{attribute 'linkalways'} 
{attribute 'no_explicit_call' := 'This FB is a CLASS and must be accessed using methods or properties'}
{attribute 'enable_dynamic_creation'}
FUNCTION_BLOCK _ETcVnFeatureScoreTypeORB EXTENDS EnumDatatypeBase
VAR
	localData : ETcVnFeatureScoreTypeORB;
	activeData : REFERENCE TO ETcVnFeatureScoreTypeORB;
	enumBaseDatatype : _DINT(localData);
END_VAR

METHOD PRIVATE AddLocalEnumeration
VAR_INPUT
	Enumeration : T_MAXSTRING;
	Value : ETcVnFeatureScoreTypeORB;
END_VAR
AddEnumeration(Enumeration, Value);
END_METHOD

PROPERTY PUBLIC Address : PVOID
GET
Address := ADR(activeData);
END_GET
END_PROPERTY

METHOD PUBLIC ClearReference
VAR_INPUT
END_VAR
activeData REF= localData;
SetBaseDatatypeReference();
END_METHOD

METHOD PUBLIC Clone : I_Datatype
VAR
    pClone : POINTER TO _ETcVnFeatureScoreTypeORB;
END_VAR
pClone := __NEW(_ETcVnFeatureScoreTypeORB(InitialValue := Value));
Clone := pClone^;
END_METHOD

METHOD FB_init : BOOL
VAR_INPUT
	bInitRetains : BOOL; // if TRUE, the retain variables are initialized (warm start / cold start)
	bInCopyCode : BOOL;  // if TRUE, the instance afterwards gets moved into the copy code (online change)
	InitialValue : ETcVnFeatureScoreTypeORB;
END_VAR
localData := InitialValue;
AddBaseDatatype(enumBaseDatatype);
ClearReference();

AddLocalEnumeration('TCVN_FST_ORB_HARRIS', ETcVnFeatureScoreTypeORB.TCVN_FST_ORB_HARRIS);
AddLocalEnumeration('TCVN_FST_ORB_FAST', ETcVnFeatureScoreTypeORB.TCVN_FST_ORB_FAST);
END_METHOD

PROPERTY PUBLIC Identifier : T_MAXSTRING
GET
Identifier := 'ETcVnFeatureScoreTypeORB';
END_GET
END_PROPERTY

METHOD IsEnumeratorValueEqual : BOOL
VAR_INPUT
	Enumerator : I_KeyValueForwardEnumerator;
END_VAR
VAR
	storedValue : ETcVnFeatureScoreTypeORB;
END_VAR
IF NOT Enumerator.TryGet(storedValue) THEN
	RETURN;
END_IF

IsEnumeratorValueEqual := storedValue = activeData;
END_METHOD

METHOD PUBLIC MakeReferenceTo
VAR_INPUT
	ReferenceTarget : REFERENCE TO ETcVnFeatureScoreTypeORB;
END_VAR
activeData REF= ReferenceTarget;
SetBaseDatatypeReference();
END_METHOD

METHOD PROTECTED SetBaseDatatypeReference
VAR_INPUT
END_VAR
enumBaseDatatype.MakeReferenceTo(activeData);
END_METHOD

PROPERTY PUBLIC Size : UDINT
GET
Size := SIZEOF(activeData);
END_GET
END_PROPERTY

METHOD TryMakeReferenceTo : BOOL
VAR_INPUT
	Target : I_Datatype;
END_VAR
VAR
	targetAsEnum : I_EnumDatatype;
	pTargetData : POINTER TO ETcVnFeatureScoreTypeORB;
END_VAR
IF NOT Target.TryResolveAsEnumDatatype(targetAsEnum) THEN
	RETURN;
END_IF

IF targetAsEnum.Identifier <> Identifier THEN
	RETURN;
END_IF

pTargetData := Target.Address;
activeData REF= pTargetData^;
SetBaseDatatypeReference();
TryMakeReferenceTo := TRUE;
END_METHOD

PROPERTY PUBLIC Value : ETcVnFeatureScoreTypeORB
GET
Value := activeData;
END_GET
SET
activeData := Value;
END_SET
END_PROPERTY

END_FUNCTION_BLOCK

(* stored: Version 1.1.0.1, ProductVersion 3.1.4024.13
   POU _ETcVnFeatureScoreTypeORB: Id {15c0cc44-f562-0f51-0f9a-718f0dddc65b}, SpecialFunc None
   Folder Core: Id {df601a09-cbae-02db-08fe-8ac88da08644}
   Folder Protected: Id {92163e21-aa89-0321-267b-a355ab4cae68}
   Folder Customize: Id {6d3a5763-e8d1-0f13-33df-945d8160b9e1}
   Folder Constructor: Id {8b40bffe-e2be-0495-1321-7413e1ad65e8}
   Folder Private: Id {aa80153e-39fb-0732-36e3-7e3ad3f38d94}
   Folder Protected: Id {4633f427-e61f-0493-0688-5742aa9f23d0}
   Method AddLocalEnumeration: Id {9f39223e-9470-039e-39a8-0675ce62e4ff}
   Property Address: Id {6760ea54-2415-03cb-3177-bfceedc2a8c9}
   Get Get: Id {5bc95193-dc58-0e53-18da-11d1bd8a60da}
   Method ClearReference: Id {e3220401-e4c1-091b-0760-324778c8aa33}
   Method Clone: Id {64985a08-8ed4-0345-30e0-1f5738597027}
   Method FB_init: Id {4c1f1c28-98dc-0ef3-3dd7-6976fc278be2}
   Property Identifier: Id {586d37b3-75d5-09d3-2f2d-6decf420cd89}
   Get Get: Id {a022818d-6baf-0e68-02ea-a5483871dd45}
   Method IsEnumeratorValueEqual: Id {2b33d57c-c436-0f53-2a77-dc3296274dcc}
   Method MakeReferenceTo: Id {a0a71ccf-1c38-0646-2fd7-83a1c69fc093}
   Method SetBaseDatatypeReference: Id {8baad4ac-5fde-0bbd-220e-99fe815f57e8}
   Property Size: Id {c0bc61ae-6c7d-0104-00af-8354506c1713}
   Get Get: Id {f22a1fa6-d1ba-0834-00c8-75cfa17030e5}
   Method TryMakeReferenceTo: Id {31401189-8d7c-030a-3ad7-e7d3ac22f4a8}
   Property Value: Id {fd167ec9-83a6-04bb-17e0-bc1cdf332d9a}
   Get Get: Id {b33305e6-e87a-0510-20d8-5a2d828aef57}
   Set Set: Id {26b25687-aed1-02eb-1af8-ae116054441a} *)
